Universal Robots PolyScope program: simplevision.urp

Program simplevision (createdIn=3.2.18654 lastSavedIn=3.2.18654 directory=/home/ur/ursim-3.2/programs/howto installation=default robotSerialNumber=2014359999)
Calibrated DH parameters: a=[0, -0.425, -0.39225, 0, 0, 0]; d=[0.089159, 0, 0, 0.10915, 0.09465, 0.0823]; alpha=[1.570796, 0, 0, 1.570796, -1.570796, 0]; deltaTheta=[0, 0, 0, 0, 0, 0]
Robot Program (runOnlyOnce=false motionType=MoveJ speed=1.047198 acceleration=1.396263 recalculateMotions=false)
  MoveJ speed 60 deg/s, acceleration 80 deg/s^2 (recalculateMotions=false)
    Waypoint refrence_point: TCP in base x=-120.113 y=-431.763 z=146.073 mm, rx=-0.0012 ry=3.1163 rz=0.0389 rad; joints [-91.713, -98.956, -126.223, -46.295, 91.393, -1.776] deg
  Folder GetCameraData Folder
    '# Here we should read the data from the camera'
    x := 100
    y := 50
    rz := 30
  Folder Calculate Folder
    '# Convert mm to m and deg to rad'
    offset := p[(x/1000), (y/1000), 0, 0, 0, d2r(rz)]
    target := pose_trans(refrence_point, offset)
  Folder MoveToCamPose
    MoveL speed 250 mm/s, acceleration 1200 mm/s^2 (recalculateMotions=false) feature=Base
      Waypoint Waypoint (Variable): variable=target
